DATA_BLOCK "ton_timer_t"
{InstructionName := 'TON';
LibVersion := '1.0';
S7_Optimized_Access := 'false' }
AUTHOR : Simatic
FAMILY : IEC_TC
NAME : TON
VERSION : 1.0
NON_RETAIN
TON

BEGIN

END_DATA_BLOCK

